// TIA Portal V20 export
DATA_BLOCK "Simulation_DB"   // DB48
// stored: InstanceOfName Unit1.Em5.Simulation, InstanceOfType FB, Namespace Unit1.Em5
"Unit1.Em5.Simulation"
   // VAR_INPUT
   //    simulation { ExternalAccessible := 'False'; ExternalVisible := 'False'; ExternalWritable := 'False'} : Bool;
   // END_VAR
   // VAR
   //    instMainPnPActuator { ExternalAccessible := 'False'; ExternalVisible := 'False'; ExternalWritable := 'False'} : Array[0..9] of "LER_SimActuator";
   //    instAlignTableActuator { ExternalAccessible := 'False'; ExternalVisible := 'False'; ExternalWritable := 'False'} : Array[0..9] of "LER_SimActuator";
   //    instNgPnPActuator { ExternalAccessible := 'False'; ExternalVisible := 'False'; ExternalWritable := 'False'} : Array[0..9] of "LER_SimActuator";
   // END_VAR
BEGIN
END_DATA_BLOCK
